TYPE IOL_2IN :
STRUCT
	BYTE0		AT %I* 	: USINT;
    BYTE1		AT %I* 	: USINT;
END_STRUCT
END_TYPE

(* stored: Version 1.1.0.1
   DUT IOL_2IN: Id {de607a47-d6ab-4aa3-bcc9-b3d20e461ab0} *)
